Fanuc KAREL source: kb00141.KL

-- PROVISIONAL review KL for V770-1; original PC SHA256 b810c842623743ee2a3a5e76f5889b97cd86a07563b4c860b6e35b1a50a46565
-- Incomplete behavior may be omitted. Consult companion uncertainty JSON. Do not deploy.
PROGRAM KB00141
%NOLOCKGROUP
BEGIN
  -- UNRESOLVED_PC offsets 5-14; opcodes 3F,75
  -- UNRESOLVED_PC offsets 19-26; opcodes 9D,23
  -- UNRESOLVED_PC offsets 31-49; opcodes 27,22,2A,22,31
  -- UNRESOLVED_PC offsets 54-58; opcodes 7F
END KB00141
